// TIA Portal V20 export
FUNCTION_BLOCK "FB_HmiKeyboardSignals"   // FB810, SCL
{ S7_Optimized_Access := 'TRUE' }
// stored: AutoNumber false, MemoryReserve 100, SetENOAutomatically false
   VAR
      sK1_Powermeter : "FB_HmiKeysSignalsManu";
      sK2_GasAssist { S7_SetPoint := 'True'} : "FB_HmiKeysSignalsManu";
      sK4a_GripperUndrilledPartClose { S7_SetPoint := 'True'} : "FB_HmiKeysSignalsManu";
      sK4b_GripperUndrilledPartOpen { S7_SetPoint := 'True'} : "FB_HmiKeysSignalsManu";
      sK5a_GripperDrilledPartClose { S7_SetPoint := 'True'} : "FB_HmiKeysSignalsManu";
      sK5b_GripperDrilledPartOpen { S7_SetPoint := 'True'} : "FB_HmiKeysSignalsManu";
      sK6_SITestStop { S7_SetPoint := 'True'} : "FB_HmiKeysSignalsManu";
      sK7_FixtureClamp { S7_SetPoint := 'True'} : "FB_HmiKeysSignalsManu";
      sK8_FixtureVacuum { S7_SetPoint := 'True'} : "FB_HmiKeysSignalsManu";
      sK9_Aspiration { S7_SetPoint := 'True'} : "FB_HmiKeysSignalsManu";
      sK12a_Backlight { S7_SetPoint := 'True'} : "FB_HmiKeysSignalsManu";
      sK12b_ObservationCamera { S7_SetPoint := 'True'} : "FB_HmiKeysSignalsManu";
      sK13_MainDoor { S7_SetPoint := 'True'} : "FB_HmiKeysSignalsManu";
      sK14_WarmUp { S7_SetPoint := 'True'} : "FB_HmiKeysSignalsManu";
      sK15_MachineLight { S7_SetPoint := 'True'} : "FB_HmiKeysSignalsManu";
   END_VAR
   VAR_TEMP
      tNoLed : Bool;   // Index for loop
   END_VAR
BEGIN
   REGION Description header 
       //==================================================================================
       // POSALUX Swiss SA / (C) Copyright 2024
       //----------------------------------------------------------------------------------
       // Title: Management of inputs and outputs for HMI buttons
       // Comment/Function: 
       //
       // Author: Fabien WALDT
       // Engineering: TIA Portal v20
       //----------------------------------------------------------------------------------
       // Change log table:
       // Version  | Date     | Expert in charge | Changes applied
       // ---------|----------|------------------|------------------------------------
       // 00.00.01 | 20251024 | WFA              | First released version
       // ==================================================================================
   END_REGION

   REGION HMI Buttons
       // K1_Powermeter 
       #sK1_Powermeter(ioOPC := "DB_OPC_Buttons".Powermeter);

       // K2_GasAssist
       #sK2_GasAssist(ioOPC := "DB_OPC_Buttons".GasAssist);

       // K4_GripperUndrilledPart
       #sK4a_GripperUndrilledPartClose(ioOPC := "DB_OPC_Buttons".GripperUndrilledClamp.Close);
       #sK4b_GripperUndrilledPartOpen(ioOPC := "DB_OPC_Buttons".GripperUndrilledClamp.Open);

       // K5_GripperDrilledPart
       #sK5a_GripperDrilledPartClose(ioOPC := "DB_OPC_Buttons".GripperDrilledClamp.Close);
       #sK5b_GripperDrilledPartOpen(ioOPC := "DB_OPC_Buttons".GripperDrilledClamp.Open);

       // K6_SITestStop
       #sK6_SITestStop(ioOPC := "DB_OPC_Buttons".SITestStop);

       // K7_FixtureClamp
       #sK7_FixtureClamp(ioOPC := "DB_OPC_Buttons".FixtureClamp);

       // K8_FixtureVacuum
       #sK8_FixtureVacuum(ioOPC := "DB_OPC_Buttons".FixtureVacuum);

       // K9_Aspiration
       #sK9_Aspiration(ioOPC := "DB_OPC_Buttons".Aspiration);

       // K12a_Backlight
       #sK12a_Backlight(ioOPC := "DB_OPC_Buttons".Backlight);

       // K12b_ObservationCamera
       #sK12b_ObservationCamera(ioOPC := "DB_OPC_Buttons".ObservationCamera);

       // K13_MainDoor
       #sK13_MainDoor(ioOPC := "DB_OPC_Buttons".MainDoor);

       // K14_WarmUp
       #sK14_WarmUp(ioOPC := "DB_OPC_Buttons".WarmUp);

       // K15_MachineLight
       #sK15_MachineLight(ioOPC := "DB_OPC_Buttons".MachineLight);
   END_REGION

   REGION Gripper
       "DB_OPC_Buttons".GripperUndrilledClamp.IsClosed := "DB_GestionGripper".sUndrilledGripper.oStateCloseWithPart OR "DB_GestionGripper".sUndrilledGripper.oStateClose;
       "DB_OPC_Buttons".GripperUndrilledClamp.IsOpened := "DB_GestionGripper".sUndrilledGripper.oStateOpen;
   END_REGION
END_FUNCTION_BLOCK
